// TIA Portal V17 export
FUNCTION "数组访问与IO标签" : Void   // FC, LAD
{ S7_Optimized_Access := 'TRUE' }
VERSION : 0.1
// stored: AutoNumber true, IsIECCheckEnabled false, SetENOAutomatically false
BEGIN

REGION Network 1
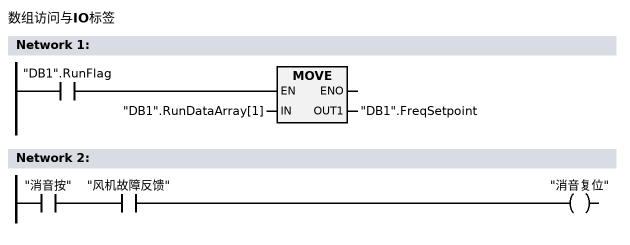
   RUNG wire#powerrail
      Contact( "DB1".RunFlag )
      { S7_GenerateENO := "TRUE" } Move(in := "DB1".RunDataArray[1], out1 => "DB1".FreqSetpoint)
   END_RUNG
   // the same network as SCL:
   IF "DB1".RunFlag THEN "DB1".FreqSetpoint := "DB1".RunDataArray[1]; END_IF;
END_REGION

REGION Network 2
   RUNG wire#powerrail
      Contact( "消音按" )
      Contact( "风机故障反馈" )
      Coil( "消音复位" )
   END_RUNG
   // the same network as SCL:
   "消音复位" := "消音按" AND "风机故障反馈";
END_REGION
END_FUNCTION
